{attribute 'linkalways'} 
{attribute 'no_explicit_call' := 'This FB is a CLASS and must be accessed using methods or properties'}
{attribute 'enable_dynamic_creation'}
FUNCTION_BLOCK InputPortChangedEvent EXTENDS Disposable IMPLEMENTS I_InputPortChangedEvent
VAR
	_targetInputPort : I_InputPort;
END_VAR

METHOD FB_init : BOOL
VAR_INPUT
	bInitRetains : BOOL; // if TRUE, the retain variables are initialized (warm start / cold start)
	bInCopyCode : BOOL;  // if TRUE, the instance afterwards gets moved into the copy code (online change)
	TargetInputPort : I_InputPort;
END_VAR
This^._targetInputPort := TargetInputPort;
END_METHOD

PROPERTY PUBLIC TargetInputPort : I_InputPort
GET
TargetInputPort := _targetInputPort;
END_GET
END_PROPERTY

END_FUNCTION_BLOCK

(* stored: Version 1.1.0.1, ProductVersion 3.1.4024.12
   POU InputPortChangedEvent: Id {5aa9e345-c5b7-074a-2401-56f7d516e868}, SpecialFunc None
   Folder Constructor: Id {6ecffc37-607f-0390-148a-cbefe941fab2}
   Method FB_init: Id {a1870d51-cc3e-0ea1-2732-7d6779f81d56}
   Property TargetInputPort: Id {3275df24-48b7-050a-1d47-fbd758ea4279}
   Get Get: Id {43c571bf-604c-06f1-3cf3-a2c29a379a21} *)
